          // MatMul: fc1
          #v3[0] := "NeuroPLC_MLP_Weights".b3[0] + "NeuroPLC_MLP_Weights".w2[0] * #v2[0] + "NeuroPLC_MLP_Weights".w2[1] * #v2[1] + "NeuroPLC_MLP_Weights".w2[2] * #v2[2] + "NeuroPLC_MLP_Weights".w2[3] * #v2[3] + "NeuroPLC_MLP_Weights".w2[4] * #v2[4] + "NeuroPLC_MLP_Weights".w2[5] * #v2[5] + "NeuroPLC_MLP_Weights".w2[6] * #v2[6] + "NeuroPLC_MLP_Weights".w2[7] * #v2[7] + "NeuroPLC_MLP_Weights".w2[8] * #v2[8] + "NeuroPLC_MLP_Weights".w2[9] * #v2[9] + "NeuroPLC_MLP_Weights".w2[10] * #v2[10] + "NeuroPLC_MLP_Weights".w2[11] * #v2[11] + "NeuroPLC_MLP_Weights".w2[12] * #v2[12] + "NeuroPLC_MLP_Weights".w2[13] * #v2[13] + "NeuroPLC_MLP_Weights".w2[14] * #v2[14] + "NeuroPLC_MLP_Weights".w2[15] * #v2[15] + "NeuroPLC_MLP_Weights".w2[16] * #v2[16] + "NeuroPLC_MLP_Weights".w2[17] * #v2[17] + "NeuroPLC_MLP_Weights".w2[18] * #v2[18] + "NeuroPLC_MLP_Weights".w2[19] * #v2[19] + "NeuroPLC_MLP_Weights".w2[20] * #v2[20] + "NeuroPLC_MLP_Weights".w2[21] * #v2[21] + "NeuroPLC_MLP_Weights".w2[22] * #v2[22] + "NeuroPLC_MLP_Weights".w2[23] * #v2[23] + "NeuroPLC_MLP_Weights".w2[24] * #v2[24] + "NeuroPLC_MLP_Weights".w2[25] * #v2[25] + "NeuroPLC_MLP_Weights".w2[26] * #v2[26] + "NeuroPLC_MLP_Weights".w2[27] * #v2[27] + "NeuroPLC_MLP_Weights".w2[28] * #v2[28] + "NeuroPLC_MLP_Weights".w2[29] * #v2[29] + "NeuroPLC_MLP_Weights".w2[30] * #v2[30] + "NeuroPLC_MLP_Weights".w2[31] * #v2[31];
          #v3[1] := "NeuroPLC_MLP_Weights".b3[1] + "NeuroPLC_MLP_Weights".w2[32] * #v2[0] + "NeuroPLC_MLP_Weights".w2[33] * #v2[1] + "NeuroPLC_MLP_Weights".w2[34] * #v2[2] + "NeuroPLC_MLP_Weights".w2[35] * #v2[3] + "NeuroPLC_MLP_Weights".w2[36] * #v2[4] + "NeuroPLC_MLP_Weights".w2[37] * #v2[5] + "NeuroPLC_MLP_Weights".w2[38] * #v2[6] + "NeuroPLC_MLP_Weights".w2[39] * #v2[7] + "NeuroPLC_MLP_Weights".w2[40] * #v2[8] + "NeuroPLC_MLP_Weights".w2[41] * #v2[9] + "NeuroPLC_MLP_Weights".w2[42] * #v2[10] + "NeuroPLC_MLP_Weights".w2[43] * #v2[11] + "NeuroPLC_MLP_Weights".w2[44] * #v2[12] + "NeuroPLC_MLP_Weights".w2[45] * #v2[13] + "NeuroPLC_MLP_Weights".w2[46] * #v2[14] + "NeuroPLC_MLP_Weights".w2[47] * #v2[15] + "NeuroPLC_MLP_Weights".w2[48] * #v2[16] + "NeuroPLC_MLP_Weights".w2[49] * #v2[17] + "NeuroPLC_MLP_Weights".w2[50] * #v2[18] + "NeuroPLC_MLP_Weights".w2[51] * #v2[19] + "NeuroPLC_MLP_Weights".w2[52] * #v2[20] + "NeuroPLC_MLP_Weights".w2[53] * #v2[21] + "NeuroPLC_MLP_Weights".w2[54] * #v2[22] + "NeuroPLC_MLP_Weights".w2[55] * #v2[23] + "NeuroPLC_MLP_Weights".w2[56] * #v2[24] + "NeuroPLC_MLP_Weights".w2[57] * #v2[25] + "NeuroPLC_MLP_Weights".w2[58] * #v2[26] + "NeuroPLC_MLP_Weights".w2[59] * #v2[27] + "NeuroPLC_MLP_Weights".w2[60] * #v2[28] + "NeuroPLC_MLP_Weights".w2[61] * #v2[29] + "NeuroPLC_MLP_Weights".w2[62] * #v2[30] + "NeuroPLC_MLP_Weights".w2[63] * #v2[31];
          #v3[2] := "NeuroPLC_MLP_Weights".b3[2] + "NeuroPLC_MLP_Weights".w2[64] * #v2[0] + "NeuroPLC_MLP_Weights".w2[65] * #v2[1] + "NeuroPLC_MLP_Weights".w2[66] * #v2[2] + "NeuroPLC_MLP_Weights".w2[67] * #v2[3] + "NeuroPLC_MLP_Weights".w2[68] * #v2[4] + "NeuroPLC_MLP_Weights".w2[69] * #v2[5] + "NeuroPLC_MLP_Weights".w2[70] * #v2[6] + "NeuroPLC_MLP_Weights".w2[71] * #v2[7] + "NeuroPLC_MLP_Weights".w2[72] * #v2[8] + "NeuroPLC_MLP_Weights".w2[73] * #v2[9] + "NeuroPLC_MLP_Weights".w2[74] * #v2[10] + "NeuroPLC_MLP_Weights".w2[75] * #v2[11] + "NeuroPLC_MLP_Weights".w2[76] * #v2[12] + "NeuroPLC_MLP_Weights".w2[77] * #v2[13] + "NeuroPLC_MLP_Weights".w2[78] * #v2[14] + "NeuroPLC_MLP_Weights".w2[79] * #v2[15] + "NeuroPLC_MLP_Weights".w2[80] * #v2[16] + "NeuroPLC_MLP_Weights".w2[81] * #v2[17] + "NeuroPLC_MLP_Weights".w2[82] * #v2[18] + "NeuroPLC_MLP_Weights".w2[83] * #v2[19] + "NeuroPLC_MLP_Weights".w2[84] * #v2[20] + "NeuroPLC_MLP_Weights".w2[85] * #v2[21] + "NeuroPLC_MLP_Weights".w2[86] * #v2[22] + "NeuroPLC_MLP_Weights".w2[87] * #v2[23] + "NeuroPLC_MLP_Weights".w2[88] * #v2[24] + "NeuroPLC_MLP_Weights".w2[89] * #v2[25] + "NeuroPLC_MLP_Weights".w2[90] * #v2[26] + "NeuroPLC_MLP_Weights".w2[91] * #v2[27] + "NeuroPLC_MLP_Weights".w2[92] * #v2[28] + "NeuroPLC_MLP_Weights".w2[93] * #v2[29] + "NeuroPLC_MLP_Weights".w2[94] * #v2[30] + "NeuroPLC_MLP_Weights".w2[95] * #v2[31];
          #v3[3] := "NeuroPLC_MLP_Weights".b3[3] + "NeuroPLC_MLP_Weights".w2[96] * #v2[0] + "NeuroPLC_MLP_Weights".w2[97] * #v2[1] + "NeuroPLC_MLP_Weights".w2[98] * #v2[2] + "NeuroPLC_MLP_Weights".w2[99] * #v2[3] + "NeuroPLC_MLP_Weights".w2[100] * #v2[4] + "NeuroPLC_MLP_Weights".w2[101] * #v2[5] + "NeuroPLC_MLP_Weights".w2[102] * #v2[6] + "NeuroPLC_MLP_Weights".w2[103] * #v2[7] + "NeuroPLC_MLP_Weights".w2[104] * #v2[8] + "NeuroPLC_MLP_Weights".w2[105] * #v2[9] + "NeuroPLC_MLP_Weights".w2[106] * #v2[10] + "NeuroPLC_MLP_Weights".w2[107] * #v2[11] + "NeuroPLC_MLP_Weights".w2[108] * #v2[12] + "NeuroPLC_MLP_Weights".w2[109] * #v2[13] + "NeuroPLC_MLP_Weights".w2[110] * #v2[14] + "NeuroPLC_MLP_Weights".w2[111] * #v2[15] + "NeuroPLC_MLP_Weights".w2[112] * #v2[16] + "NeuroPLC_MLP_Weights".w2[113] * #v2[17] + "NeuroPLC_MLP_Weights".w2[114] * #v2[18] + "NeuroPLC_MLP_Weights".w2[115] * #v2[19] + "NeuroPLC_MLP_Weights".w2[116] * #v2[20] + "NeuroPLC_MLP_Weights".w2[117] * #v2[21] + "NeuroPLC_MLP_Weights".w2[118] * #v2[22] + "NeuroPLC_MLP_Weights".w2[119] * #v2[23] + "NeuroPLC_MLP_Weights".w2[120] * #v2[24] + "NeuroPLC_MLP_Weights".w2[121] * #v2[25] + "NeuroPLC_MLP_Weights".w2[122] * #v2[26] + "NeuroPLC_MLP_Weights".w2[123] * #v2[27] + "NeuroPLC_MLP_Weights".w2[124] * #v2[28] + "NeuroPLC_MLP_Weights".w2[125] * #v2[29] + "NeuroPLC_MLP_Weights".w2[126] * #v2[30] + "NeuroPLC_MLP_Weights".w2[127] * #v2[31];
          #v3[4] := "NeuroPLC_MLP_Weights".b3[4] + "NeuroPLC_MLP_Weights".w2[128] * #v2[0] + "NeuroPLC_MLP_Weights".w2[129] * #v2[1] + "NeuroPLC_MLP_Weights".w2[130] * #v2[2] + "NeuroPLC_MLP_Weights".w2[131] * #v2[3] + "NeuroPLC_MLP_Weights".w2[132] * #v2[4] + "NeuroPLC_MLP_Weights".w2[133] * #v2[5] + "NeuroPLC_MLP_Weights".w2[134] * #v2[6] + "NeuroPLC_MLP_Weights".w2[135] * #v2[7] + "NeuroPLC_MLP_Weights".w2[136] * #v2[8] + "NeuroPLC_MLP_Weights".w2[137] * #v2[9] + "NeuroPLC_MLP_Weights".w2[138] * #v2[10] + "NeuroPLC_MLP_Weights".w2[139] * #v2[11] + "NeuroPLC_MLP_Weights".w2[140] * #v2[12] + "NeuroPLC_MLP_Weights".w2[141] * #v2[13] + "NeuroPLC_MLP_Weights".w2[142] * #v2[14] + "NeuroPLC_MLP_Weights".w2[143] * #v2[15] + "NeuroPLC_MLP_Weights".w2[144] * #v2[16] + "NeuroPLC_MLP_Weights".w2[145] * #v2[17] + "NeuroPLC_MLP_Weights".w2[146] * #v2[18] + "NeuroPLC_MLP_Weights".w2[147] * #v2[19] + "NeuroPLC_MLP_Weights".w2[148] * #v2[20] + "NeuroPLC_MLP_Weights".w2[149] * #v2[21] + "NeuroPLC_MLP_Weights".w2[150] * #v2[22] + "NeuroPLC_MLP_Weights".w2[151] * #v2[23] + "NeuroPLC_MLP_Weights".w2[152] * #v2[24] + "NeuroPLC_MLP_Weights".w2[153] * #v2[25] + "NeuroPLC_MLP_Weights".w2[154] * #v2[26] + "NeuroPLC_MLP_Weights".w2[155] * #v2[27] + "NeuroPLC_MLP_Weights".w2[156] * #v2[28] + "NeuroPLC_MLP_Weights".w2[157] * #v2[29] + "NeuroPLC_MLP_Weights".w2[158] * #v2[30] + "NeuroPLC_MLP_Weights".w2[159] * #v2[31];
          #v3[5] := "NeuroPLC_MLP_Weights".b3[5] + "NeuroPLC_MLP_Weights".w2[160] * #v2[0] + "NeuroPLC_MLP_Weights".w2[161] * #v2[1] + "NeuroPLC_MLP_Weights".w2[162] * #v2[2] + "NeuroPLC_MLP_Weights".w2[163] * #v2[3] + "NeuroPLC_MLP_Weights".w2[164] * #v2[4] + "NeuroPLC_MLP_Weights".w2[165] * #v2[5] + "NeuroPLC_MLP_Weights".w2[166] * #v2[6] + "NeuroPLC_MLP_Weights".w2[167] * #v2[7] + "NeuroPLC_MLP_Weights".w2[168] * #v2[8] + "NeuroPLC_MLP_Weights".w2[169] * #v2[9] + "NeuroPLC_MLP_Weights".w2[170] * #v2[10] + "NeuroPLC_MLP_Weights".w2[171] * #v2[11] + "NeuroPLC_MLP_Weights".w2[172] * #v2[12] + "NeuroPLC_MLP_Weights".w2[173] * #v2[13] + "NeuroPLC_MLP_Weights".w2[174] * #v2[14] + "NeuroPLC_MLP_Weights".w2[175] * #v2[15] + "NeuroPLC_MLP_Weights".w2[176] * #v2[16] + "NeuroPLC_MLP_Weights".w2[177] * #v2[17] + "NeuroPLC_MLP_Weights".w2[178] * #v2[18] + "NeuroPLC_MLP_Weights".w2[179] * #v2[19] + "NeuroPLC_MLP_Weights".w2[180] * #v2[20] + "NeuroPLC_MLP_Weights".w2[181] * #v2[21] + "NeuroPLC_MLP_Weights".w2[182] * #v2[22] + "NeuroPLC_MLP_Weights".w2[183] * #v2[23] + "NeuroPLC_MLP_Weights".w2[184] * #v2[24] + "NeuroPLC_MLP_Weights".w2[185] * #v2[25] + "NeuroPLC_MLP_Weights".w2[186] * #v2[26] + "NeuroPLC_MLP_Weights".w2[187] * #v2[27] + "NeuroPLC_MLP_Weights".w2[188] * #v2[28] + "NeuroPLC_MLP_Weights".w2[189] * #v2[29] + "NeuroPLC_MLP_Weights".w2[190] * #v2[30] + "NeuroPLC_MLP_Weights".w2[191] * #v2[31];
          #v3[6] := "NeuroPLC_MLP_Weights".b3[6] + "NeuroPLC_MLP_Weights".w2[192] * #v2[0] + "NeuroPLC_MLP_Weights".w2[193] * #v2[1] + "NeuroPLC_MLP_Weights".w2[194] * #v2[2] + "NeuroPLC_MLP_Weights".w2[195] * #v2[3] + "NeuroPLC_MLP_Weights".w2[196] * #v2[4] + "NeuroPLC_MLP_Weights".w2[197] * #v2[5] + "NeuroPLC_MLP_Weights".w2[198] * #v2[6] + "NeuroPLC_MLP_Weights".w2[199] * #v2[7] + "NeuroPLC_MLP_Weights".w2[200] * #v2[8] + "NeuroPLC_MLP_Weights".w2[201] * #v2[9] + "NeuroPLC_MLP_Weights".w2[202] * #v2[10] + "NeuroPLC_MLP_Weights".w2[203] * #v2[11] + "NeuroPLC_MLP_Weights".w2[204] * #v2[12] + "NeuroPLC_MLP_Weights".w2[205] * #v2[13] + "NeuroPLC_MLP_Weights".w2[206] * #v2[14] + "NeuroPLC_MLP_Weights".w2[207] * #v2[15] + "NeuroPLC_MLP_Weights".w2[208] * #v2[16] + "NeuroPLC_MLP_Weights".w2[209] * #v2[17] + "NeuroPLC_MLP_Weights".w2[210] * #v2[18] + "NeuroPLC_MLP_Weights".w2[211] * #v2[19] + "NeuroPLC_MLP_Weights".w2[212] * #v2[20] + "NeuroPLC_MLP_Weights".w2[213] * #v2[21] + "NeuroPLC_MLP_Weights".w2[214] * #v2[22] + "NeuroPLC_MLP_Weights".w2[215] * #v2[23] + "NeuroPLC_MLP_Weights".w2[216] * #v2[24] + "NeuroPLC_MLP_Weights".w2[217] * #v2[25] + "NeuroPLC_MLP_Weights".w2[218] * #v2[26] + "NeuroPLC_MLP_Weights".w2[219] * #v2[27] + "NeuroPLC_MLP_Weights".w2[220] * #v2[28] + "NeuroPLC_MLP_Weights".w2[221] * #v2[29] + "NeuroPLC_MLP_Weights".w2[222] * #v2[30] + "NeuroPLC_MLP_Weights".w2[223] * #v2[31];
          #v3[7] := "NeuroPLC_MLP_Weights".b3[7] + "NeuroPLC_MLP_Weights".w2[224] * #v2[0] + "NeuroPLC_MLP_Weights".w2[225] * #v2[1] + "NeuroPLC_MLP_Weights".w2[226] * #v2[2] + "NeuroPLC_MLP_Weights".w2[227] * #v2[3] + "NeuroPLC_MLP_Weights".w2[228] * #v2[4] + "NeuroPLC_MLP_Weights".w2[229] * #v2[5] + "NeuroPLC_MLP_Weights".w2[230] * #v2[6] + "NeuroPLC_MLP_Weights".w2[231] * #v2[7] + "NeuroPLC_MLP_Weights".w2[232] * #v2[8] + "NeuroPLC_MLP_Weights".w2[233] * #v2[9] + "NeuroPLC_MLP_Weights".w2[234] * #v2[10] + "NeuroPLC_MLP_Weights".w2[235] * #v2[11] + "NeuroPLC_MLP_Weights".w2[236] * #v2[12] + "NeuroPLC_MLP_Weights".w2[237] * #v2[13] + "NeuroPLC_MLP_Weights".w2[238] * #v2[14] + "NeuroPLC_MLP_Weights".w2[239] * #v2[15] + "NeuroPLC_MLP_Weights".w2[240] * #v2[16] + "NeuroPLC_MLP_Weights".w2[241] * #v2[17] + "NeuroPLC_MLP_Weights".w2[242] * #v2[18] + "NeuroPLC_MLP_Weights".w2[243] * #v2[19] + "NeuroPLC_MLP_Weights".w2[244] * #v2[20] + "NeuroPLC_MLP_Weights".w2[245] * #v2[21] + "NeuroPLC_MLP_Weights".w2[246] * #v2[22] + "NeuroPLC_MLP_Weights".w2[247] * #v2[23] + "NeuroPLC_MLP_Weights".w2[248] * #v2[24] + "NeuroPLC_MLP_Weights".w2[249] * #v2[25] + "NeuroPLC_MLP_Weights".w2[250] * #v2[26] + "NeuroPLC_MLP_Weights".w2[251] * #v2[27] + "NeuroPLC_MLP_Weights".w2[252] * #v2[28] + "NeuroPLC_MLP_Weights".w2[253] * #v2[29] + "NeuroPLC_MLP_Weights".w2[254] * #v2[30] + "NeuroPLC_MLP_Weights".w2[255] * #v2[31];
          #v3[8] := "NeuroPLC_MLP_Weights".b3[8] + "NeuroPLC_MLP_Weights".w2[256] * #v2[0] + "NeuroPLC_MLP_Weights".w2[257] * #v2[1] + "NeuroPLC_MLP_Weights".w2[258] * #v2[2] + "NeuroPLC_MLP_Weights".w2[259] * #v2[3] + "NeuroPLC_MLP_Weights".w2[260] * #v2[4] + "NeuroPLC_MLP_Weights".w2[261] * #v2[5] + "NeuroPLC_MLP_Weights".w2[262] * #v2[6] + "NeuroPLC_MLP_Weights".w2[263] * #v2[7] + "NeuroPLC_MLP_Weights".w2[264] * #v2[8] + "NeuroPLC_MLP_Weights".w2[265] * #v2[9] + "NeuroPLC_MLP_Weights".w2[266] * #v2[10] + "NeuroPLC_MLP_Weights".w2[267] * #v2[11] + "NeuroPLC_MLP_Weights".w2[268] * #v2[12] + "NeuroPLC_MLP_Weights".w2[269] * #v2[13] + "NeuroPLC_MLP_Weights".w2[270] * #v2[14] + "NeuroPLC_MLP_Weights".w2[271] * #v2[15] + "NeuroPLC_MLP_Weights".w2[272] * #v2[16] + "NeuroPLC_MLP_Weights".w2[273] * #v2[17] + "NeuroPLC_MLP_Weights".w2[274] * #v2[18] + "NeuroPLC_MLP_Weights".w2[275] * #v2[19] + "NeuroPLC_MLP_Weights".w2[276] * #v2[20] + "NeuroPLC_MLP_Weights".w2[277] * #v2[21] + "NeuroPLC_MLP_Weights".w2[278] * #v2[22] + "NeuroPLC_MLP_Weights".w2[279] * #v2[23] + "NeuroPLC_MLP_Weights".w2[280] * #v2[24] + "NeuroPLC_MLP_Weights".w2[281] * #v2[25] + "NeuroPLC_MLP_Weights".w2[282] * #v2[26] + "NeuroPLC_MLP_Weights".w2[283] * #v2[27] + "NeuroPLC_MLP_Weights".w2[284] * #v2[28] + "NeuroPLC_MLP_Weights".w2[285] * #v2[29] + "NeuroPLC_MLP_Weights".w2[286] * #v2[30] + "NeuroPLC_MLP_Weights".w2[287] * #v2[31];
          #v3[9] := "NeuroPLC_MLP_Weights".b3[9] + "NeuroPLC_MLP_Weights".w2[288] * #v2[0] + "NeuroPLC_MLP_Weights".w2[289] * #v2[1] + "NeuroPLC_MLP_Weights".w2[290] * #v2[2] + "NeuroPLC_MLP_Weights".w2[291] * #v2[3] + "NeuroPLC_MLP_Weights".w2[292] * #v2[4] + "NeuroPLC_MLP_Weights".w2[293] * #v2[5] + "NeuroPLC_MLP_Weights".w2[294] * #v2[6] + "NeuroPLC_MLP_Weights".w2[295] * #v2[7] + "NeuroPLC_MLP_Weights".w2[296] * #v2[8] + "NeuroPLC_MLP_Weights".w2[297] * #v2[9] + "NeuroPLC_MLP_Weights".w2[298] * #v2[10] + "NeuroPLC_MLP_Weights".w2[299] * #v2[11] + "NeuroPLC_MLP_Weights".w2[300] * #v2[12] + "NeuroPLC_MLP_Weights".w2[301] * #v2[13] + "NeuroPLC_MLP_Weights".w2[302] * #v2[14] + "NeuroPLC_MLP_Weights".w2[303] * #v2[15] + "NeuroPLC_MLP_Weights".w2[304] * #v2[16] + "NeuroPLC_MLP_Weights".w2[305] * #v2[17] + "NeuroPLC_MLP_Weights".w2[306] * #v2[18] + "NeuroPLC_MLP_Weights".w2[307] * #v2[19] + "NeuroPLC_MLP_Weights".w2[308] * #v2[20] + "NeuroPLC_MLP_Weights".w2[309] * #v2[21] + "NeuroPLC_MLP_Weights".w2[310] * #v2[22] + "NeuroPLC_MLP_Weights".w2[311] * #v2[23] + "NeuroPLC_MLP_Weights".w2[312] * #v2[24] + "NeuroPLC_MLP_Weights".w2[313] * #v2[25] + "NeuroPLC_MLP_Weights".w2[314] * #v2[26] + "NeuroPLC_MLP_Weights".w2[315] * #v2[27] + "NeuroPLC_MLP_Weights".w2[316] * #v2[28] + "NeuroPLC_MLP_Weights".w2[317] * #v2[29] + "NeuroPLC_MLP_Weights".w2[318] * #v2[30] + "NeuroPLC_MLP_Weights".w2[319] * #v2[31];
          #v3[10] := "NeuroPLC_MLP_Weights".b3[10] + "NeuroPLC_MLP_Weights".w2[320] * #v2[0] + "NeuroPLC_MLP_Weights".w2[321] * #v2[1] + "NeuroPLC_MLP_Weights".w2[322] * #v2[2] + "NeuroPLC_MLP_Weights".w2[323] * #v2[3] + "NeuroPLC_MLP_Weights".w2[324] * #v2[4] + "NeuroPLC_MLP_Weights".w2[325] * #v2[5] + "NeuroPLC_MLP_Weights".w2[326] * #v2[6] + "NeuroPLC_MLP_Weights".w2[327] * #v2[7] + "NeuroPLC_MLP_Weights".w2[328] * #v2[8] + "NeuroPLC_MLP_Weights".w2[329] * #v2[9] + "NeuroPLC_MLP_Weights".w2[330] * #v2[10] + "NeuroPLC_MLP_Weights".w2[331] * #v2[11] + "NeuroPLC_MLP_Weights".w2[332] * #v2[12] + "NeuroPLC_MLP_Weights".w2[333] * #v2[13] + "NeuroPLC_MLP_Weights".w2[334] * #v2[14] + "NeuroPLC_MLP_Weights".w2[335] * #v2[15] + "NeuroPLC_MLP_Weights".w2[336] * #v2[16] + "NeuroPLC_MLP_Weights".w2[337] * #v2[17] + "NeuroPLC_MLP_Weights".w2[338] * #v2[18] + "NeuroPLC_MLP_Weights".w2[339] * #v2[19] + "NeuroPLC_MLP_Weights".w2[340] * #v2[20] + "NeuroPLC_MLP_Weights".w2[341] * #v2[21] + "NeuroPLC_MLP_Weights".w2[342] * #v2[22] + "NeuroPLC_MLP_Weights".w2[343] * #v2[23] + "NeuroPLC_MLP_Weights".w2[344] * #v2[24] + "NeuroPLC_MLP_Weights".w2[345] * #v2[25] + "NeuroPLC_MLP_Weights".w2[346] * #v2[26] + "NeuroPLC_MLP_Weights".w2[347] * #v2[27] + "NeuroPLC_MLP_Weights".w2[348] * #v2[28] + "NeuroPLC_MLP_Weights".w2[349] * #v2[29] + "NeuroPLC_MLP_Weights".w2[350] * #v2[30] + "NeuroPLC_MLP_Weights".w2[351] * #v2[31];
          #v3[11] := "NeuroPLC_MLP_Weights".b3[11] + "NeuroPLC_MLP_Weights".w2[352] * #v2[0] + "NeuroPLC_MLP_Weights".w2[353] * #v2[1] + "NeuroPLC_MLP_Weights".w2[354] * #v2[2] + "NeuroPLC_MLP_Weights".w2[355] * #v2[3] + "NeuroPLC_MLP_Weights".w2[356] * #v2[4] + "NeuroPLC_MLP_Weights".w2[357] * #v2[5] + "NeuroPLC_MLP_Weights".w2[358] * #v2[6] + "NeuroPLC_MLP_Weights".w2[359] * #v2[7] + "NeuroPLC_MLP_Weights".w2[360] * #v2[8] + "NeuroPLC_MLP_Weights".w2[361] * #v2[9] + "NeuroPLC_MLP_Weights".w2[362] * #v2[10] + "NeuroPLC_MLP_Weights".w2[363] * #v2[11] + "NeuroPLC_MLP_Weights".w2[364] * #v2[12] + "NeuroPLC_MLP_Weights".w2[365] * #v2[13] + "NeuroPLC_MLP_Weights".w2[366] * #v2[14] + "NeuroPLC_MLP_Weights".w2[367] * #v2[15] + "NeuroPLC_MLP_Weights".w2[368] * #v2[16] + "NeuroPLC_MLP_Weights".w2[369] * #v2[17] + "NeuroPLC_MLP_Weights".w2[370] * #v2[18] + "NeuroPLC_MLP_Weights".w2[371] * #v2[19] + "NeuroPLC_MLP_Weights".w2[372] * #v2[20] + "NeuroPLC_MLP_Weights".w2[373] * #v2[21] + "NeuroPLC_MLP_Weights".w2[374] * #v2[22] + "NeuroPLC_MLP_Weights".w2[375] * #v2[23] + "NeuroPLC_MLP_Weights".w2[376] * #v2[24] + "NeuroPLC_MLP_Weights".w2[377] * #v2[25] + "NeuroPLC_MLP_Weights".w2[378] * #v2[26] + "NeuroPLC_MLP_Weights".w2[379] * #v2[27] + "NeuroPLC_MLP_Weights".w2[380] * #v2[28] + "NeuroPLC_MLP_Weights".w2[381] * #v2[29] + "NeuroPLC_MLP_Weights".w2[382] * #v2[30] + "NeuroPLC_MLP_Weights".w2[383] * #v2[31];
          #v3[12] := "NeuroPLC_MLP_Weights".b3[12] + "NeuroPLC_MLP_Weights".w2[384] * #v2[0] + "NeuroPLC_MLP_Weights".w2[385] * #v2[1] + "NeuroPLC_MLP_Weights".w2[386] * #v2[2] + "NeuroPLC_MLP_Weights".w2[387] * #v2[3] + "NeuroPLC_MLP_Weights".w2[388] * #v2[4] + "NeuroPLC_MLP_Weights".w2[389] * #v2[5] + "NeuroPLC_MLP_Weights".w2[390] * #v2[6] + "NeuroPLC_MLP_Weights".w2[391] * #v2[7] + "NeuroPLC_MLP_Weights".w2[392] * #v2[8] + "NeuroPLC_MLP_Weights".w2[393] * #v2[9] + "NeuroPLC_MLP_Weights".w2[394] * #v2[10] + "NeuroPLC_MLP_Weights".w2[395] * #v2[11] + "NeuroPLC_MLP_Weights".w2[396] * #v2[12] + "NeuroPLC_MLP_Weights".w2[397] * #v2[13] + "NeuroPLC_MLP_Weights".w2[398] * #v2[14] + "NeuroPLC_MLP_Weights".w2[399] * #v2[15] + "NeuroPLC_MLP_Weights".w2[400] * #v2[16] + "NeuroPLC_MLP_Weights".w2[401] * #v2[17] + "NeuroPLC_MLP_Weights".w2[402] * #v2[18] + "NeuroPLC_MLP_Weights".w2[403] * #v2[19] + "NeuroPLC_MLP_Weights".w2[404] * #v2[20] + "NeuroPLC_MLP_Weights".w2[405] * #v2[21] + "NeuroPLC_MLP_Weights".w2[406] * #v2[22] + "NeuroPLC_MLP_Weights".w2[407] * #v2[23] + "NeuroPLC_MLP_Weights".w2[408] * #v2[24] + "NeuroPLC_MLP_Weights".w2[409] * #v2[25] + "NeuroPLC_MLP_Weights".w2[410] * #v2[26] + "NeuroPLC_MLP_Weights".w2[411] * #v2[27] + "NeuroPLC_MLP_Weights".w2[412] * #v2[28] + "NeuroPLC_MLP_Weights".w2[413] * #v2[29] + "NeuroPLC_MLP_Weights".w2[414] * #v2[30] + "NeuroPLC_MLP_Weights".w2[415] * #v2[31];
          #v3[13] := "NeuroPLC_MLP_Weights".b3[13] + "NeuroPLC_MLP_Weights".w2[416] * #v2[0] + "NeuroPLC_MLP_Weights".w2[417] * #v2[1] + "NeuroPLC_MLP_Weights".w2[418] * #v2[2] + "NeuroPLC_MLP_Weights".w2[419] * #v2[3] + "NeuroPLC_MLP_Weights".w2[420] * #v2[4] + "NeuroPLC_MLP_Weights".w2[421] * #v2[5] + "NeuroPLC_MLP_Weights".w2[422] * #v2[6] + "NeuroPLC_MLP_Weights".w2[423] * #v2[7] + "NeuroPLC_MLP_Weights".w2[424] * #v2[8] + "NeuroPLC_MLP_Weights".w2[425] * #v2[9] + "NeuroPLC_MLP_Weights".w2[426] * #v2[10] + "NeuroPLC_MLP_Weights".w2[427] * #v2[11] + "NeuroPLC_MLP_Weights".w2[428] * #v2[12] + "NeuroPLC_MLP_Weights".w2[429] * #v2[13] + "NeuroPLC_MLP_Weights".w2[430] * #v2[14] + "NeuroPLC_MLP_Weights".w2[431] * #v2[15] + "NeuroPLC_MLP_Weights".w2[432] * #v2[16] + "NeuroPLC_MLP_Weights".w2[433] * #v2[17] + "NeuroPLC_MLP_Weights".w2[434] * #v2[18] + "NeuroPLC_MLP_Weights".w2[435] * #v2[19] + "NeuroPLC_MLP_Weights".w2[436] * #v2[20] + "NeuroPLC_MLP_Weights".w2[437] * #v2[21] + "NeuroPLC_MLP_Weights".w2[438] * #v2[22] + "NeuroPLC_MLP_Weights".w2[439] * #v2[23] + "NeuroPLC_MLP_Weights".w2[440] * #v2[24] + "NeuroPLC_MLP_Weights".w2[441] * #v2[25] + "NeuroPLC_MLP_Weights".w2[442] * #v2[26] + "NeuroPLC_MLP_Weights".w2[443] * #v2[27] + "NeuroPLC_MLP_Weights".w2[444] * #v2[28] + "NeuroPLC_MLP_Weights".w2[445] * #v2[29] + "NeuroPLC_MLP_Weights".w2[446] * #v2[30] + "NeuroPLC_MLP_Weights".w2[447] * #v2[31];
          #v3[14] := "NeuroPLC_MLP_Weights".b3[14] + "NeuroPLC_MLP_Weights".w2[448] * #v2[0] + "NeuroPLC_MLP_Weights".w2[449] * #v2[1] + "NeuroPLC_MLP_Weights".w2[450] * #v2[2] + "NeuroPLC_MLP_Weights".w2[451] * #v2[3] + "NeuroPLC_MLP_Weights".w2[452] * #v2[4] + "NeuroPLC_MLP_Weights".w2[453] * #v2[5] + "NeuroPLC_MLP_Weights".w2[454] * #v2[6] + "NeuroPLC_MLP_Weights".w2[455] * #v2[7] + "NeuroPLC_MLP_Weights".w2[456] * #v2[8] + "NeuroPLC_MLP_Weights".w2[457] * #v2[9] + "NeuroPLC_MLP_Weights".w2[458] * #v2[10] + "NeuroPLC_MLP_Weights".w2[459] * #v2[11] + "NeuroPLC_MLP_Weights".w2[460] * #v2[12] + "NeuroPLC_MLP_Weights".w2[461] * #v2[13] + "NeuroPLC_MLP_Weights".w2[462] * #v2[14] + "NeuroPLC_MLP_Weights".w2[463] * #v2[15] + "NeuroPLC_MLP_Weights".w2[464] * #v2[16] + "NeuroPLC_MLP_Weights".w2[465] * #v2[17] + "NeuroPLC_MLP_Weights".w2[466] * #v2[18] + "NeuroPLC_MLP_Weights".w2[467] * #v2[19] + "NeuroPLC_MLP_Weights".w2[468] * #v2[20] + "NeuroPLC_MLP_Weights".w2[469] * #v2[21] + "NeuroPLC_MLP_Weights".w2[470] * #v2[22] + "NeuroPLC_MLP_Weights".w2[471] * #v2[23] + "NeuroPLC_MLP_Weights".w2[472] * #v2[24] + "NeuroPLC_MLP_Weights".w2[473] * #v2[25] + "NeuroPLC_MLP_Weights".w2[474] * #v2[26] + "NeuroPLC_MLP_Weights".w2[475] * #v2[27] + "NeuroPLC_MLP_Weights".w2[476] * #v2[28] + "NeuroPLC_MLP_Weights".w2[477] * #v2[29] + "NeuroPLC_MLP_Weights".w2[478] * #v2[30] + "NeuroPLC_MLP_Weights".w2[479] * #v2[31];
          #v3[15] := "NeuroPLC_MLP_Weights".b3[15] + "NeuroPLC_MLP_Weights".w2[480] * #v2[0] + "NeuroPLC_MLP_Weights".w2[481] * #v2[1] + "NeuroPLC_MLP_Weights".w2[482] * #v2[2] + "NeuroPLC_MLP_Weights".w2[483] * #v2[3] + "NeuroPLC_MLP_Weights".w2[484] * #v2[4] + "NeuroPLC_MLP_Weights".w2[485] * #v2[5] + "NeuroPLC_MLP_Weights".w2[486] * #v2[6] + "NeuroPLC_MLP_Weights".w2[487] * #v2[7] + "NeuroPLC_MLP_Weights".w2[488] * #v2[8] + "NeuroPLC_MLP_Weights".w2[489] * #v2[9] + "NeuroPLC_MLP_Weights".w2[490] * #v2[10] + "NeuroPLC_MLP_Weights".w2[491] * #v2[11] + "NeuroPLC_MLP_Weights".w2[492] * #v2[12] + "NeuroPLC_MLP_Weights".w2[493] * #v2[13] + "NeuroPLC_MLP_Weights".w2[494] * #v2[14] + "NeuroPLC_MLP_Weights".w2[495] * #v2[15] + "NeuroPLC_MLP_Weights".w2[496] * #v2[16] + "NeuroPLC_MLP_Weights".w2[497] * #v2[17] + "NeuroPLC_MLP_Weights".w2[498] * #v2[18] + "NeuroPLC_MLP_Weights".w2[499] * #v2[19] + "NeuroPLC_MLP_Weights".w2[500] * #v2[20] + "NeuroPLC_MLP_Weights".w2[501] * #v2[21] + "NeuroPLC_MLP_Weights".w2[502] * #v2[22] + "NeuroPLC_MLP_Weights".w2[503] * #v2[23] + "NeuroPLC_MLP_Weights".w2[504] * #v2[24] + "NeuroPLC_MLP_Weights".w2[505] * #v2[25] + "NeuroPLC_MLP_Weights".w2[506] * #v2[26] + "NeuroPLC_MLP_Weights".w2[507] * #v2[27] + "NeuroPLC_MLP_Weights".w2[508] * #v2[28] + "NeuroPLC_MLP_Weights".w2[509] * #v2[29] + "NeuroPLC_MLP_Weights".w2[510] * #v2[30] + "NeuroPLC_MLP_Weights".w2[511] * #v2[31];

          // StandardAct: relu
          FOR #i := 0 TO 15 DO
              IF #v3[#i] < 0.0 THEN
                  #v4[#i] := 0.0;
              ELSE
                  #v4[#i] := #v3[#i];
              END_IF;
          END_FOR;

          // MatMul: fc2
          #v5[0] := "NeuroPLC_MLP_Weights".b5[0] + "NeuroPLC_MLP_Weights".w4[0] * #v4[0] + "NeuroPLC_MLP_Weights".w4[1] * #v4[1] + "NeuroPLC_MLP_Weights".w4[2] * #v4[2] + "NeuroPLC_MLP_Weights".w4[3] * #v4[3] + "NeuroPLC_MLP_Weights".w4[4] * #v4[4] + "NeuroPLC_MLP_Weights".w4[5] * #v4[5] + "NeuroPLC_MLP_Weights".w4[6] * #v4[6] + "NeuroPLC_MLP_Weights".w4[7] * #v4[7] + "NeuroPLC_MLP_Weights".w4[8] * #v4[8] + "NeuroPLC_MLP_Weights".w4[9] * #v4[9] + "NeuroPLC_MLP_Weights".w4[10] * #v4[10] + "NeuroPLC_MLP_Weights".w4[11] * #v4[11] + "NeuroPLC_MLP_Weights".w4[12] * #v4[12] + "NeuroPLC_MLP_Weights".w4[13] * #v4[13] + "NeuroPLC_MLP_Weights".w4[14] * #v4[14] + "NeuroPLC_MLP_Weights".w4[15] * #v4[15];
          #v5[1] := "NeuroPLC_MLP_Weights".b5[1] + "NeuroPLC_MLP_Weights".w4[16] * #v4[0] + "NeuroPLC_MLP_Weights".w4[17] * #v4[1] + "NeuroPLC_MLP_Weights".w4[18] * #v4[2] + "NeuroPLC_MLP_Weights".w4[19] * #v4[3] + "NeuroPLC_MLP_Weights".w4[20] * #v4[4] + "NeuroPLC_MLP_Weights".w4[21] * #v4[5] + "NeuroPLC_MLP_Weights".w4[22] * #v4[6] + "NeuroPLC_MLP_Weights".w4[23] * #v4[7] + "NeuroPLC_MLP_Weights".w4[24] * #v4[8] + "NeuroPLC_MLP_Weights".w4[25] * #v4[9] + "NeuroPLC_MLP_Weights".w4[26] * #v4[10] + "NeuroPLC_MLP_Weights".w4[27] * #v4[11] + "NeuroPLC_MLP_Weights".w4[28] * #v4[12] + "NeuroPLC_MLP_Weights".w4[29] * #v4[13] + "NeuroPLC_MLP_Weights".w4[30] * #v4[14] + "NeuroPLC_MLP_Weights".w4[31] * #v4[15];
          #v5[2] := "NeuroPLC_MLP_Weights".b5[2] + "NeuroPLC_MLP_Weights".w4[32] * #v4[0] + "NeuroPLC_MLP_Weights".w4[33] * #v4[1] + "NeuroPLC_MLP_Weights".w4[34] * #v4[2] + "NeuroPLC_MLP_Weights".w4[35] * #v4[3] + "NeuroPLC_MLP_Weights".w4[36] * #v4[4] + "NeuroPLC_MLP_Weights".w4[37] * #v4[5] + "NeuroPLC_MLP_Weights".w4[38] * #v4[6] + "NeuroPLC_MLP_Weights".w4[39] * #v4[7] + "NeuroPLC_MLP_Weights".w4[40] * #v4[8] + "NeuroPLC_MLP_Weights".w4[41] * #v4[9] + "NeuroPLC_MLP_Weights".w4[42] * #v4[10] + "NeuroPLC_MLP_Weights".w4[43] * #v4[11] + "NeuroPLC_MLP_Weights".w4[44] * #v4[12] + "NeuroPLC_MLP_Weights".w4[45] * #v4[13] + "NeuroPLC_MLP_Weights".w4[46] * #v4[14] + "NeuroPLC_MLP_Weights".w4[47] * #v4[15];
          #v5[3] := "NeuroPLC_MLP_Weights".b5[3] + "NeuroPLC_MLP_Weights".w4[48] * #v4[0] + "NeuroPLC_MLP_Weights".w4[49] * #v4[1] + "NeuroPLC_MLP_Weights".w4[50] * #v4[2] + "NeuroPLC_MLP_Weights".w4[51] * #v4[3] + "NeuroPLC_MLP_Weights".w4[52] * #v4[4] + "NeuroPLC_MLP_Weights".w4[53] * #v4[5] + "NeuroPLC_MLP_Weights".w4[54] * #v4[6] + "NeuroPLC_MLP_Weights".w4[55] * #v4[7] + "NeuroPLC_MLP_Weights".w4[56] * #v4[8] + "NeuroPLC_MLP_Weights".w4[57] * #v4[9] + "NeuroPLC_MLP_Weights".w4[58] * #v4[10] + "NeuroPLC_MLP_Weights".w4[59] * #v4[11] + "NeuroPLC_MLP_Weights".w4[60] * #v4[12] + "NeuroPLC_MLP_Weights".w4[61] * #v4[13] + "NeuroPLC_MLP_Weights".w4[62] * #v4[14] + "NeuroPLC_MLP_Weights".w4[63] * #v4[15];

          // Softmax
          #max_val := #v5[0];
          FOR #i := 1 TO 3 DO
              IF #v5[#i] > #max_val THEN
                  #max_val := #v5[#i];
              END_IF;
          END_FOR;
          #sum := 0.0;
          FOR #i := 0 TO 3 DO
              #v6[#i] := EXP(#v5[#i] - #max_val);
              #sum := #sum + #v6[#i];
          END_FOR;
          FOR #i := 0 TO 3 DO
              #v6[#i] := #v6[#i] / #sum;
          END_FOR;

          // Argmax
          #max_val := #v6[0];
          #fault_class := 0;
          FOR #i := 1 TO 3 DO
              IF #v6[#i] > #max_val THEN
                  #max_val := #v6[#i];
                  #fault_class := #i;
              END_IF;
          END_FOR;
          #confidence := #max_val;
END_FUNCTION_BLOCK

ORGANIZATION_BLOCK "Main"   // OB1, LAD, ProgramCycle
TITLE = "Main Program Sweep (Cycle)"
{ S7_Optimized_Access := 'TRUE' }
VERSION : 0.1
   VAR_INPUT
      Initial_Call : Bool;   // Initial call of this OB
      Remanence : Bool;   // =True, if remanent data are available
   END_VAR
BEGIN
END_ORGANIZATION_BLOCK